{attribute 'GeneratedUsingTerminal: EK1122-0000-0018'}
{attribute addProperty BoxType "EK1122-0000-0018"}
{attribute addProperty Id "Beckhoff_ER3xxxsub_EK1100EK1100_1FC0878B2A_0001_ER3174_0002_0016ER3174_DCC7866252A_0002_ER3174_0002_0022ER3174_DCC7866252A_0003_ER3174_0002_0023ER3174_DCC7866252A_0004_ER3184_0002_0019ER3184_DCC7866252A_0005_ER3184_0002_0020ER3184_DCC7866252A_0006_ER3184_0002_0021ER3184_DCC7866252A_0007_ER3184_1002_0020ER3184_DCC7866252A_0008_ER3184_1002_0021ER3184_DCC7866252A_0009_ER3204_0002_0016ER3204_6CD7E11952A_0010_ER3204_0002_0020ER3204_6CD7E11952A_0011_ER3204_0002_0021ER3204_5380707048A_0012_ER3314_0002_0021ER3314_B654D23048"}
{attribute addProperty CRC "1812749530"}
{attribute addProperty Size "618"}
TYPE Beckhoff_ER3xxxEK1122_6C0C5CDA EXTENDS EK1122_1FC0878B :
STRUCT
	{attribute addProperty Name "Beckhoff_ER3xxxsub_EK1100"}
	Beckhoff_ER3xxxsub_EK1100 : EK1100_1FC0878B;
	{attribute addProperty Name "A_0001_ER3174_0002_0016"}
	A_0001_ER3174_0002_0016 : ER3174_DCC78662;
	{attribute addProperty Name "A_0002_ER3174_0002_0022"}
	A_0002_ER3174_0002_0022 : ER3174_DCC78662;
	{attribute addProperty Name "A_0003_ER3174_0002_0023"}
	A_0003_ER3174_0002_0023 : ER3174_DCC78662;
	{attribute addProperty Name "A_0004_ER3184_0002_0019"}
	A_0004_ER3184_0002_0019 : ER3184_DCC78662;
	{attribute addProperty Name "A_0005_ER3184_0002_0020"}
	A_0005_ER3184_0002_0020 : ER3184_DCC78662;
	{attribute addProperty Name "A_0006_ER3184_0002_0021"}
	A_0006_ER3184_0002_0021 : ER3184_DCC78662;
	{attribute addProperty Name "A_0007_ER3184_1002_0020"}
	A_0007_ER3184_1002_0020 : ER3184_DCC78662;
	{attribute addProperty Name "A_0008_ER3184_1002_0021"}
	A_0008_ER3184_1002_0021 : ER3184_DCC78662;
	{attribute addProperty Name "A_0009_ER3204_0002_0016"}
	A_0009_ER3204_0002_0016 : ER3204_6CD7E119;
	{attribute addProperty Name "A_0010_ER3204_0002_0020"}
	A_0010_ER3204_0002_0020 : ER3204_6CD7E119;
	{attribute addProperty Name "A_0011_ER3204_0002_0021"}
	A_0011_ER3204_0002_0021 : ER3204_53807070;
	{attribute addProperty Name "A_0012_ER3314_0002_0021"}
	A_0012_ER3314_0002_0021 : ER3314_B654D230;
END_STRUCT
END_TYPE

(* stored: Version 1.2.0.0, ProductVersion 3.1.4024.9
   DUT Beckhoff_ER3xxxEK1122_6C0C5CDA: Id {5c487626-61ea-458e-b212-b9e4f065d7a6} *)
